INTERFACE IVtemByFesto

METHOD moveBwd : BOOL
VAR_INPUT
END_VAR
END_METHOD

METHOD moveFwd : BOOL
VAR_INPUT
END_VAR
END_METHOD

END_INTERFACE

(* stored: Version 1.1.0.1, ProductVersion 3.1.4024.12
   Itf IVtemByFesto: Id {c671ce13-b39c-446e-a6e3-c4670dc09ad1}
   Method moveBwd: Id {dc1cb979-4985-4f25-8434-a885560df841}
   Method moveFwd: Id {4d09c024-2fdf-4efc-995c-96559d768b1e} *)
